FUNCTION TIME_TO_REAL (* SPEZIAL-Hilfsfunktion dieses Projekts (NICHT Teil der echten OSCAT_basic-Konvertierungsbibliothek, KEIN Standard-IEC-61131-3-Block) - liefert TM als REAL in Millisekunden (UDINT_TO_REAL(TIME_IN_MS_TO_UDINT(TM))). Trotz generischem Namen beim Suchen/Portieren nicht mit einem echten Standardblock verwechseln. *)
  (* Standard: 61499-1 *)
  (* Version 1.0, 2025-12-21, Franz Höpfinger, Eigene Hilfsfunktion, nicht aus OSCAT_basic portiert - liefert TIME als REAL-Millisekunden. Franz (2026-09-17, nach Verwechslungsgefahr bei der FT_PT1-Portierung): 'TIME_TO_REAL gibt es nicht... aaaaaaaaaaaaaah SPEZIAL' - dieser Kommentar/Remark soll genau diese Verwechslung kuenftig verhindern. *)
  PACKAGE OSCAT::Basic::POUs::conversion;
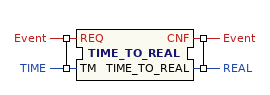
  EVENT_INPUT
    REQ WITH TM;
  END_EVENT
  EVENT_OUTPUT
    CNF WITH TIME_TO_REAL;
  END_EVENT
  VAR_INPUT
    TM : TIME;
  END_VAR
  VAR_OUTPUT
    TIME_TO_REAL : REAL;
  END_VAR
  BODY IN ST:
PACKAGE OSCAT::Basic::POUs::conversion;

FUNCTION TIME_TO_REAL : REAL
VAR_INPUT
	TM : TIME;
END_VAR

TIME_TO_REAL := UDINT_TO_REAL(TIME_IN_MS_TO_UDINT(TM));

END_FUNCTION
  END_BODY
END_FUNCTION
